FUNCTION_BLOCK FB_Roboterablauf
VAR_INPUT
	bEnable : BOOL;
	bExecute : BOOL;
END_VAR
VAR_OUTPUT
	eState : eBetriebszustand;
END_VAR
VAR
	nState : INT := 0;
	nStation : INT := 1;
	nFlaschenPos : INT := 1;
	fbRobotersteuerung : FB_Robotersteuerung;
	fbTon : TON;
END_VAR

fbRobotersteuerung(
	bEnable:= , 
	bExecute:= , 
	rXpos:= , 
	rYpos:= , 
	rZpos:= , 
	bGclose:= , 
	eState=> );
	
fbTon(IN:= , PT:= T#5S, Q=> , ET=> );
	
CASE nState OF
	0: // OFF
	eState := eBetriebszustand.OFF;
	
	fbRobotersteuerung.bEnable := FALSE;
	
	IF bEnable THEN
		nState := 1;
	END_IF
	
	1: // INIT
	eState := eBetriebszustand.INIT;
	
	fbRobotersteuerung.bEnable := TRUE;
	
	IF fbRobotersteuerung.eState = eBetriebszustand.READY THEN
		nState := 2;
	END_IF
	
	2: // INIT - HomePos
	eState := eBetriebszustand.INIT;
	
	fbRobotersteuerung.rXpos := GVL_PosKinematic.pXhome;
	fbRobotersteuerung.rYpos := GVL_PosKinematic.pYhome;
	fbRobotersteuerung.rZpos := GVL_PosKinematic.pYhome;
	fbRobotersteuerung.bGclose := FALSE;
	fbRobotersteuerung.bExecute := TRUE;
	
	IF fbRobotersteuerung.eState = eBetriebszustand.READY THEN
		fbRobotersteuerung.bExecute := FALSE;
		nState := 3;
	END_IF
	
	3: // READY
	eState := eBetriebszustand.READY;
	
	IF bExecute THEN
		nState := 4;
	END_IF
	
	4: // PROD - PickUp
	eState := eBetriebszustand.PROD;
	
	fbRobotersteuerung.rXpos := GVL_PosKinematic.pXconv;
	fbRobotersteuerung.rYpos := GVL_PosKinematic.pYconv;
	fbRobotersteuerung.rZpos := GVL_PosKinematic.pZconv;
	fbRobotersteuerung.bGclose := TRUE;
	fbRobotersteuerung.bExecute := TRUE;
	fbTon.IN := TRUE;
	IF fbTon.Q THEN nStation := 2; END_IF
	
	IF fbRobotersteuerung.eState = eBetriebszustand.DONE
		AND nStation = 2 THEN
		fbTon.IN := FALSE;
		fbRobotersteuerung.bExecute := FALSE;
		nState := 5;
	END_IF
	
	5: // PROD - Waage
	eState := eBetriebszustand.PROD;
	
	fbRobotersteuerung.rXpos := GVL_PosKinematic.pXscale;
	fbRobotersteuerung.rYpos := GVL_PosKinematic.pYscale;
	fbRobotersteuerung.rZpos := GVL_PosKinematic.pZscale;
	fbRobotersteuerung.bGclose := TRUE;
	fbRobotersteuerung.bExecute := TRUE;
	fbTon.IN := TRUE;
	IF fbTon.Q THEN nStation := 3; END_IF
	
	IF fbRobotersteuerung.eState = eBetriebszustand.DONE 
		AND nStation = 3 THEN
		fbTon.IN := FALSE;
		fbRobotersteuerung.bExecute := FALSE;
		nState := 6;
	END_IF
	
	6: // PROD - Ofen
	eState := eBetriebszustand.PROD;
	
	fbRobotersteuerung.rXpos := GVL_PosKinematic.pXheat;
	fbRobotersteuerung.rYpos := GVL_PosKinematic.pYheat;
	fbRobotersteuerung.rZpos := GVL_PosKinematic.pZheat;
	fbRobotersteuerung.bGclose := TRUE;
	fbRobotersteuerung.bExecute := TRUE;
	fbTon.IN := TRUE;
	IF fbTon.Q THEN nStation := 4; END_IF
	
	IF fbRobotersteuerung.eState = eBetriebszustand.DONE 
		AND nStation = 4 THEN
		fbTon.IN := FALSE;
		fbRobotersteuerung.bExecute := FALSE;
		nState := 7;
	END_IF
	
	7: // PROD - Place
	eState := eBetriebszustand.PROD;
	
	CASE nFlaschenPos OF
	1: fbRobotersteuerung.rXpos := GVL_PosKinematic.pX1stor;
	2: fbRobotersteuerung.rXpos := GVL_PosKinematic.pX2stor;
	3: fbRobotersteuerung.rXpos := GVL_PosKinematic.pX3stor;
	4: fbRobotersteuerung.rXpos := GVL_PosKinematic.pX4stor;
	END_CASE
	fbRobotersteuerung.rYpos := GVL_PosKinematic.pYstor;
	fbRobotersteuerung.rZpos := GVL_PosKinematic.pZstor;
	fbRobotersteuerung.bGclose := FALSE;
	fbRobotersteuerung.bExecute := TRUE;
	fbTon.IN := TRUE;
	IF fbTon.Q THEN nStation := 5; END_IF
	
	IF fbRobotersteuerung.eState = eBetriebszustand.DONE
		AND nStation = 5 THEN
		fbTon.IN := FALSE;
		fbRobotersteuerung.bExecute := FALSE;
		nFlaschenPos := (nFlaschenPos MOD 4) + 1;
		nState := 8;
	END_IF
	
	8: // INIT - HomePos
	eState := eBetriebszustand.INIT;
	
	fbRobotersteuerung.rXpos := GVL_PosKinematic.pXhome;
	fbRobotersteuerung.rYpos := GVL_PosKinematic.pYhome;
	fbRobotersteuerung.rZpos := GVL_PosKinematic.pZhome;
	fbRobotersteuerung.bGclose := FALSE;
	fbRobotersteuerung.bExecute := TRUE;
	fbTon.IN := TRUE;
	IF fbTon.Q THEN nStation := 6; END_IF
	
	IF fbRobotersteuerung.eState = eBetriebszustand.DONE
		AND nStation = 6 THEN
		fbTon.IN := FALSE;
		fbRobotersteuerung.bExecute := FALSE;
		nState := 9;
	END_IF
	
	9: // DONE
	eState := eBetriebszustand.DONE;
	
	IF NOT bExecute	THEN
		fbRobotersteuerung.bExecute := FALSE;
		nState := 3;
	END_IF
	
	
END_CASE

END_FUNCTION_BLOCK

(* stored: Version 1.1.0.1, ProductVersion 3.1.4024.15
   POU FB_Roboterablauf: Id {9caf7aa8-aeaf-40c6-b498-9ccabc82f656}, SpecialFunc None *)
